FUNCTION_BLOCK Calculator IMPLEMENTS ISum

METHOD Sum : DINT
VAR_INPUT
	Dint1 : DINT;
	Dint2 : DINT;
END_VAR
Sum := Dint1 + Dint2;
END_METHOD

END_FUNCTION_BLOCK

(* stored: Version 1.1.0.1, ProductVersion 3.1.4024.6
   POU Calculator: Id {38feb073-ce6b-4189-971d-839f619c1a28}, SpecialFunc None
   Method Sum: Id {86933668-06b7-48b0-a6b4-659d968eedae} *)
